FUNCTION_BLOCK Process
VAR_INPUT
	ixInc:BOOL;
	ixDec:BOOL;
END_VAR
VAR_OUTPUT
	qxCurrentPos:INT;
	qxPosA:BOOL;
	qxPosB:BOOL;
END_VAR
VAR
END_VAR

IF ixInc AND qxCurrentPos<486 THEN
	qxCurrentPos:= qxCurrentPos + 1;
ELSIF ixDec AND qxCurrentPos>0 THEN
	qxCurrentPos:= qxCurrentPos - 1;
END_IF

IF qxCurrentPos = 486 THEN
	qxPosB:= TRUE;
ELSIF qxCurrentPos = 0 THEN
	qxPosA:= TRUE;
ELSE
	qxPosB:= FALSE;
	qxPosA:= FALSE;
END_IF

END_FUNCTION_BLOCK

(* stored: Version 1.1.0.1, ProductVersion 3.1.4024.12
   POU Process: Id {2fccb5d1-ce4a-47a7-bc58-2a6f5bfd27d0}, SpecialFunc None *)
